FUNCTION F_GetElementOrders : ST_FunctionOrders
(**************************************************************************************
 * 	Application		:	BoxControl Framework
 *	Revision		:	$Revision: 404529 $
 *	Revision date	:	$Date: 2018-04-23 08:21:38 +0200 (Mo., 23 Apr 2018) $
 *	Last changed by	:	$Author: b7bolm $
 *	URL				:	$URL: http://almscdc.swisslog.com/repo/SWPD/Development/BoxControlFramework/20_Release/trunk/01_Software/BCF/BCF/JumpStart/20_Product/10_App/13_Elements/10_Lib/10_Conv/10_Functions/F_GetElementOrders.TcPOU $
 *
 *	Purpose			:	Returns function order data
 *
 * ------------------------------------------------------------------------------------
 *	Copyright Swisslog [IP AG], Switzerland. All rights reserved.
 * 
 * ------------------------------------------------------------------------------------
 *	
 * 	Revision History: 
 *
 * 	VERSION			DATE			INITIALS			DESCRIPTION
 *	0.1				01.01.2001		swl					Example
 *
 **************************************************************************************)
VAR_INPUT
	eFunctionNumber		: E_FunctionNumber; // Function number
END_VAR


// Check if function number is valid
IF eFunctionNumber > E_FunctionNumber.F_BEGIN_FUNCTION AND
   eFunctionNumber < E_FunctionNumber.F_END_FUNCTION THEN
   
	IF __ISVALIDREF(FunctionRegistry[eFunctionNumber].rFunctionInterface) THEN
		// Return element orders
		F_GetElementOrders := FunctionRegistry[eFunctionNumber].rFunctionInterface.Out.FunctionOrders;
	END_IF
END_IF

END_FUNCTION

(* stored: Version 1.1.0.1, ProductVersion 3.1.4022.12
   POU F_GetElementOrders: Id {cdbfa8b3-2987-4b7f-b338-35057f88fb12}, SpecialFunc None *)
